// TIA Portal V17 export
// export: Created 2025-07-17T00:36:37.9178638Z, ExportSetting WithDefaults, DisplayName Totally Integrated Automation Portal, DisplayVersion V17, DisplayName TIA Portal Openness, DisplayVersion V17, DisplayName TIA Portal Version Control Interface, DisplayVersion V17, DisplayName STEP 7 Professional, DisplayVersion V17, DisplayName STEP 7 Safety, DisplayVersion V17, DisplayName WinCC Advanced / Unified PC, DisplayVersion V17
FUNCTION_BLOCK "pump_start_stop"   // FB1, LAD
{ S7_Optimized_Access := 'TRUE' }
VERSION : 0.1
// stored: AutoNumber true, IsIECCheckEnabled false, IsRetainMemResEnabled false, MemoryReserve 100, SetENOAutomatically false, UDAEnableTagReadback false
   VAR_INPUT
      tank_valve_1 : Bool;
      tank_valve_2 : Bool;
      start_stop_local : Bool;
      start_stop_remote : Bool;
      maintain : Bool;
      pump_error : Bool;
      local_remote : Bool;
      emergency_stop : Bool;
   END_VAR
   VAR_OUTPUT
      start_stop_action : Bool;
   END_VAR
BEGIN

REGION Network 1
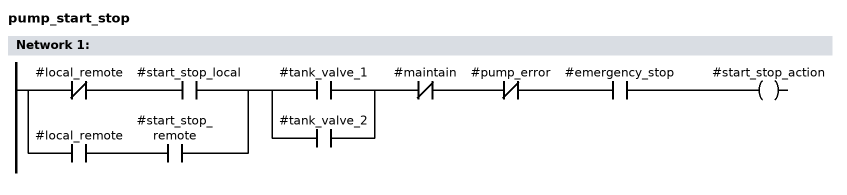
   RUNG wire#powerrail
      I_Contact( #local_remote )
      Contact( #start_stop_local )
      wire#w1
      Contact( #tank_valve_1 )
      wire#w2
      I_Contact( #maintain )
      I_Contact( #pump_error )
      Contact( #emergency_stop )
      Coil( #start_stop_action )
   END_RUNG
   RUNG wire#powerrail
      Contact( #local_remote )
      Contact( #start_stop_remote )
   END_RUNG wire#w1
   RUNG wire#w1
      Contact( #tank_valve_2 )
   END_RUNG wire#w2
   // the same network as SCL:
   #start_stop_action := ((NOT #local_remote AND #start_stop_local) OR (#local_remote AND #start_stop_remote)) AND (#tank_valve_1 OR #tank_valve_2) AND NOT #maintain AND NOT #pump_error AND #emergency_stop;
END_REGION
END_FUNCTION_BLOCK
